INTERFACE IInput

METHOD GetInputData : EngelInputData
END_METHOD

END_INTERFACE

(* stored: Version 1.1.0.1, ProductVersion 3.1.4024.12
   Itf IInput: Id {e2ee5310-5cba-4699-ae4a-a08130a9dc68}
   Method GetInputData: Id {69eef123-16ab-40f6-adc0-b1e8482bfcb4} *)
